// Mitsubishi GX Works2 project: 시퀀스 전체 반복 회로 (카운터)   PLC: Q03UDV

PROGRAM MAIN
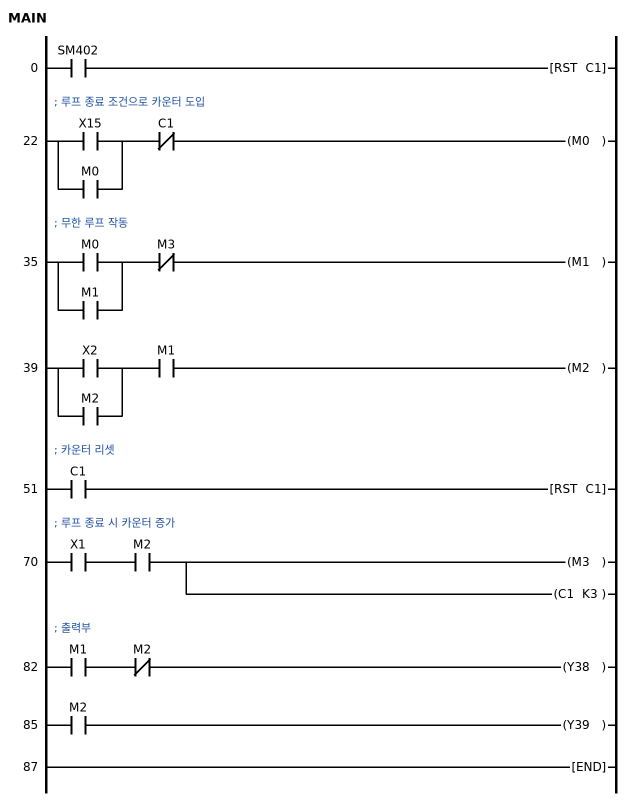
0     LD      SM402
      RST     C1
; 루프 종료 조건으로 카운터 도입
22    LD      X15
      OR      M0
      ANI     C1
      OUT     M0
; 무한 루프 작동
35    LD      M0
      OR      M1
      ANI     M3
      OUT     M1
39    LD      X2
      OR      M2
      AND     M1
      OUT     M2
; 카운터 리셋
51    LD      C1
      RST     C1
; 루프 종료 시 카운터 증가
70    LD      X1
      AND     M2
      OUT     M3
      OUT     C1 K3
; 출력부
82    LD      M1
      ANI     M2
      OUT     Y38
85    LD      M2
      OUT     Y39
87    END
END_PROGRAM
